TYPE ST_GantryErrors :
STRUCT
	Collision					: BOOL;
	EndLimitHorFront			: BOOL;
	EndLimitHorBack				: BOOL;
	EndLimitVertUp				: BOOL;
	EndLimitVertDown			: BOOL;
	ProductLost					: ARRAY [1..6] OF BOOL;
	
	VerticalNCAxisError			: ST_NcAxis_Errors;
	HorizontalNCAxisError		: ST_NcAxis_Errors;
END_STRUCT
END_TYPE

(* stored: Version 1.1.0.1, ProductVersion 3.1.4020.12
   DUT ST_GantryErrors: Id {01cf582a-17dd-4229-b88a-99184135fecd} *)
